Universal Robots PolyScope program: RC_E1_PLACE_130.urp

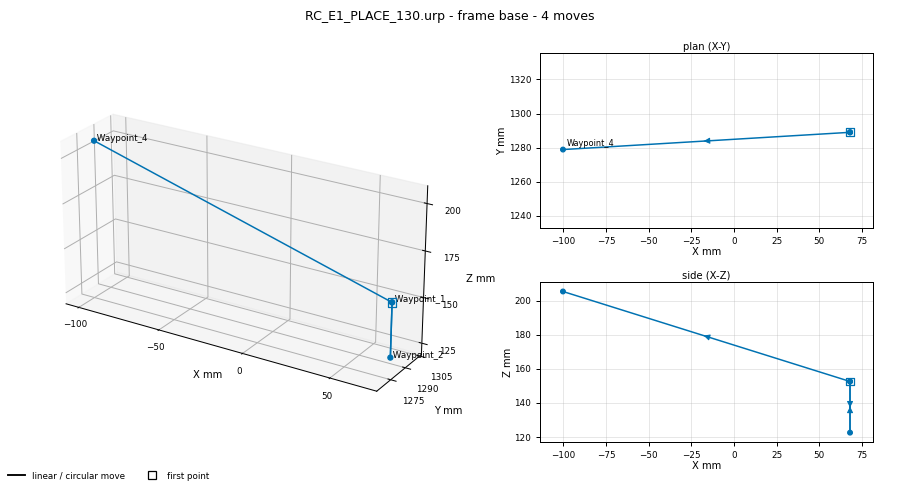
[picture p0: tool path of RC_E1_PLACE_130.urp in frame base, 4 of 4 moves have a stored position in this frame; points joined in program order, loops and branches not executed]
Program RC_E1_PLACE_130 (createdIn=3.0.0 lastSavedIn=3.0.0 directory=/programs installation=default)
Robot Program (runOnlyOnce=true motionType=MoveJ speed=1.047198 acceleration=1.396263 useActiveTCP=false)
  'Program generated by RoboDK v4.1.0 for UR3e_HORNO on 05/09/2022 13:29:59'
  'Using nominal kinematics.'
  'Using Ref. Frame No Ok 03: p[-0.386000, 1.280000, -0.011500, 0.000000, 0.000000, 0.000000]'
  'Using TCP 0208-0001-0001-307-000-3 Horno: p[0.000000, 0.000000, 0.164750, 0.000000, 0.000000, 0.000000]'
  Script: set_tcp(p[0.000000, 0.000000, 0.164750, 0.000000, 0.000000, 0.000000])
  Script: movej([0.488640, -1.452680, -1.300990, -1.967374, 1.554986, 0.448862],0.60000,0.12500,0,0.0000)
  MoveL speed 100 mm/s, acceleration 120 mm/s^2 (useActiveTCP=true)
    Waypoint Waypoint_1: TCP in base x=68 y=1289 z=152.609 mm, rx=-2.2241 ry=2.2133 rz=0.0278 rad; joints [17.321, -129.541, -27.949, -112.792, 90.999, 17.041] deg; flange x=69.631 y=1286.5 z=317.332 mm, rx=-2.2241 ry=2.2133 rz=0.0278 rad
    Waypoint Waypoint_2: TCP in base x=68 y=1289 z=122.609 mm, rx=-2.2241 ry=2.2133 rz=0.0278 rad; joints [17.321, -125.971, -42.578, -101.734, 90.999, 17.041] deg; flange x=69.631 y=1286.5 z=287.332 mm, rx=-2.2241 ry=2.2133 rz=0.0278 rad
  'Detach from 0208-0001-0001-307-000-3 Horno'
  MoveL speed 500 mm/s, acceleration 900 mm/s^2 (useActiveTCP=true)
    Waypoint Waypoint_3: TCP in base x=68 y=1289 z=152.609 mm, rx=-2.2241 ry=2.2133 rz=0.0278 rad; joints [17.321, -129.541, -27.949, -112.792, 90.999, 17.041] deg; flange x=69.631 y=1286.5 z=317.332 mm, rx=-2.2241 ry=2.2133 rz=0.0278 rad
    Waypoint Waypoint_4: TCP in base x=-100.259 y=1278.894 z=205.352 mm, rx=2.2557 ry=-2.1676 rz=0.0193 rad; joints [27.997, -83.232, -74.541, -112.722, 89.094, 25.718] deg; flange x=-100.223 y=1281.863 z=370.076 mm, rx=2.2557 ry=-2.1676 rz=0.0193 rad
